PROGRAM ILC
VAR
	e_new: LREAL;
	
END_VAR

IF LernenFertig = FALSE THEN
	e_new := GlobaleVariablen.Sollkraft - GlobaleVariablen.Fadenzugkraft_2;
	IF (e_new < (GlobaleVariablen.Sollkraft - 1)) OR (e_new > (GlobaleVariablen.Sollkraft + 1)) THEN
		u_new := u_Old[k] - 0.2 * e_new;
	ELSIF (e_new >= (GlobaleVariablen.Sollkraft - 1)) AND (e_new <= (GlobaleVariablen.Sollkraft + 1)) THEN
		u_new := u_Old[k];
	END_IF
	//PRG_MovingAverage_1();// Moving Average Filter
	
	//Verwendung der "heutigen Daten" als Steuersignal
	ILC_Out := u_new;
	IF ABS(alt_xPunkt) > 180 AND ABS(alt_xPunkt) <= 400 THEN
		IF ILC_Out>0 THEN
			ILC_Out := 0;
		ELSIF ILC_Out < 0 AND  ILC_Out < -2 * e_new THEN
			ILC_Out := -2 * e_new;
		END_IF
	ELSIF ABS(alt_xPunkt) > 400 THEN
		IF ILC_Out>0 AND ILC_Out > - 0.5*e_new THEN
			ILC_Out := - 0.5*e_new;
		ELSIF ILC_Out < 0 AND  ILC_Out < -2 * e_new THEN
			ILC_Out := -2 * e_new;
		END_IF
	END_IF
	
	//"heutige Daten" als "alte Daten" sperchern
	u_Old[k] := ILC_Out;
	e_Old[k] := e_new;
	
	IF ABS(alt_xPunkt) <= 180 THEN
		IF ABS(e_new) > 1 THEN
			LernenFertig := FALSE;
			count := 0;
		ELSE 
			count := count + 1;
		END_IF 
		
		IF count >= 1999 THEN
			LernenFertig := TRUE;
		END_IF
		
	ELSIF ABS(alt_xPunkt) > 180 AND ABS(alt_xPunkt) <= 400 THEN
		IF ABS(e_new) > 2 THEN
			LernenFertig := FALSE;
			count := 0;
		ELSE 
			count := count + 1;
		END_IF 
		
		IF count >= 1999 THEN
			LernenFertig := TRUE;
		END_IF
	ELSIF ABS(alt_xPunkt) > 400 THEN
		IF ABS(e_new) > 4 THEN
			LernenFertig := FALSE;
			count := 0;
		ELSE 
			count := count + 1;
		END_IF 
		
		IF count >= 1999 THEN
			LernenFertig := TRUE;
		END_IF
	END_IF
ELSE
	ILC_Out := u_Old[k];
END_IF

IF ABS(alt_xPunkt) <= 180 THEN
	IF ABS(GlobaleVariablen.Sollkraft - GlobaleVariablen.Fadenzugkraft_2) > 1 THEN
		LernenFertig := FALSE;
	END_IF
ELSIF ABS(alt_xPunkt) > 180 AND ABS(alt_xPunkt) <= 400 THEN
	IF ABS(GlobaleVariablen.Sollkraft - GlobaleVariablen.Fadenzugkraft_2) > 2.3 THEN
		LernenFertig := FALSE;
	END_IF
ELSIF ABS(alt_xPunkt) > 400 THEN
	IF ABS(GlobaleVariablen.Sollkraft - GlobaleVariablen.Fadenzugkraft_2) > 4 THEN
		LernenFertig := FALSE;
	END_IF
END_IF

END_PROGRAM

(* stored: Version 1.1.0.1, ProductVersion 3.1.4024.11
   POU ILC: Id {a9bae5d1-b9ee-4137-9da3-6e167f6894bd}, SpecialFunc None *)
